// TIA Portal V16 export
// export: Created 2024-03-27T10:00:42.3648579Z, ExportSetting WithDefaults, DisplayName Totally Integrated Automation Portal, DisplayVersion V16, DisplayName TIA Portal Version Control Interface, DisplayVersion V16, DisplayName TIA Portal Openness, DisplayVersion V16, DisplayName STEP 7 Professional, DisplayVersion V16, DisplayName STEP 7 Safety, DisplayVersion V16, DisplayName WinCC Advanced, DisplayVersion V16
TYPE "UR_2_T2O_IO"
// stored: IsFailsafeCompliant false
   STRUCT
      IOs { S7_SetPoint := 'True'} : "UR__T2O_IOs";
      Tool { S7_SetPoint := 'True'} : "UR__T2O_Tool";
   END_STRUCT;
END_TYPE
